// TIA Portal V17 export
// export: Created 2025-03-07T09:19:10.5525524Z, ExportSetting WithDefaults, DisplayName Totally Integrated Automation Portal, DisplayVersion V17 Update 8, DisplayName TIA Portal Openness, DisplayVersion V17 Update 8, DisplayName TIA Portal Version Control Interface, DisplayVersion V17, DisplayName SINAMICS Startdrive Advanced, DisplayVersion V17 SP2, DisplayName SINAMICS Startdrive G110M, G120, G120C, G120D, G120P, G115D, DisplayVersion V17 SP2, DisplayName SINAMICS Startdrive G130, G150, S120, S150, SINAMICS MV, S210, DisplayVersion V17 SP2, DisplayName STEP 7 Professional, DisplayVersion V17 Update 8, DisplayName SINUMERIK ONE STEP 7 Toolbox, DisplayVersion V17 Update 12, DisplayName SINUMERIK 840D sl STEP 7 Toolbox, DisplayVersion V17 Update 12, DisplayName STEP 7 Safety, DisplayVersion V17 Update 6, DisplayName WinCC Advanced, DisplayVersion V17 Update 8
FUNCTION "FC7201_HMI_DATA_FUNC" : Void   // FC7201, LAD
{ S7_Optimized_Access := 'FALSE' }
AUTHOR : ETXETAR
VERSION : 1.0
// stored: AutoNumber false, IsIECCheckEnabled false, SetENOAutomatically false, UDAEnableTagReadback false
   VAR_TEMP
      Sammel_1 : Bool;
      Sammel_2 : Bool;
      Sammel_3 : Bool;
      pin_main_table : Bool;
      main_table : Bool;
      Status1 : Int;
      Status2 : Int;
      sammel : Bool;
      aux1 : Bool;
      aux2 : Bool;
   END_VAR
   VAR_TEMP   // added for the SCL form of the ladder/FBD networks
      _w1 : Bool;
   END_VAR
BEGIN

REGION Network 1: AUTOMATIC
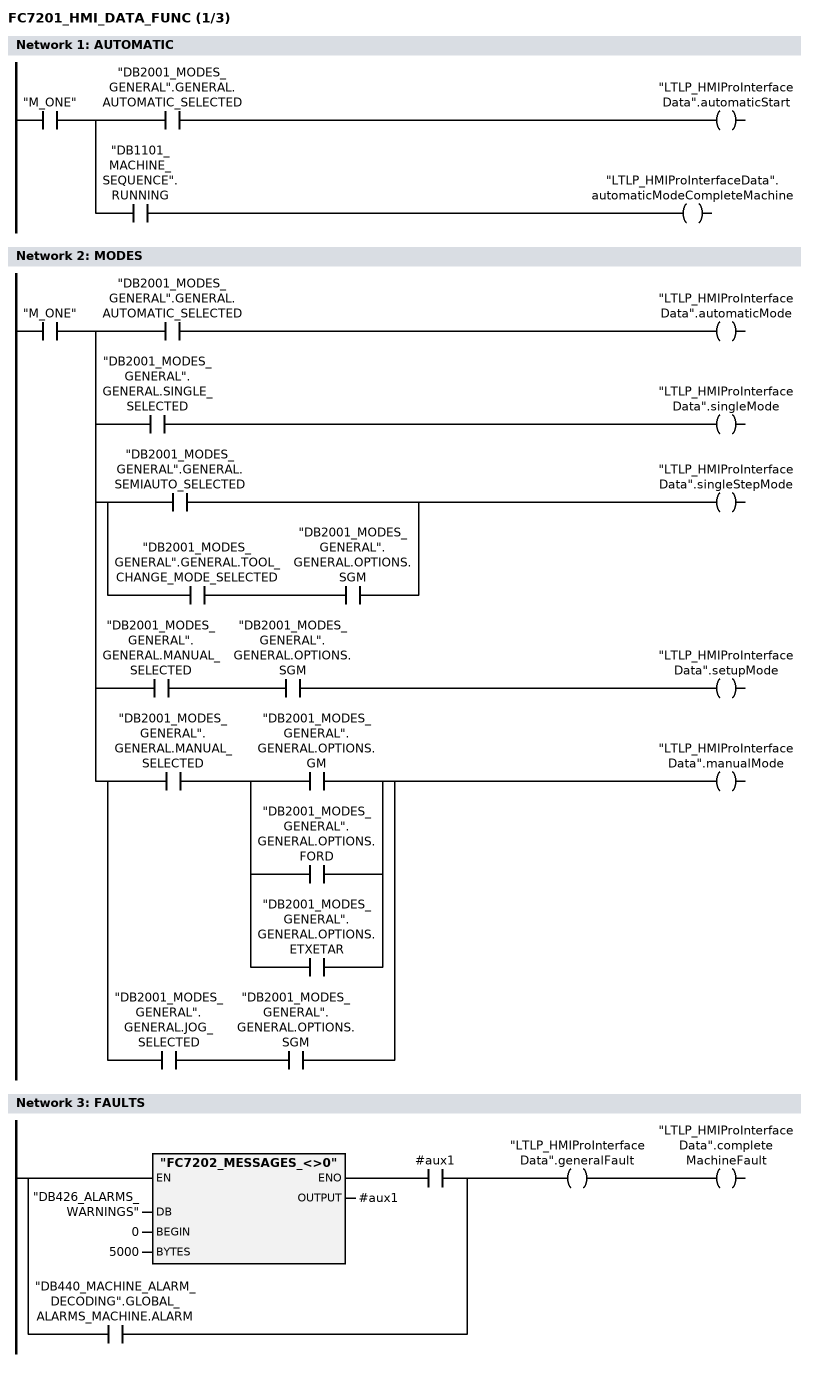
   RUNG wire#powerrail
      Contact( "M_ONE" )
      wire#w1
      Contact( "DB2001_MODES_GENERAL".GENERAL.AUTOMATIC_SELECTED )
      Coil( "LTLP_HMIProInterfaceData".automaticStart )
   END_RUNG
   RUNG wire#w1
      Contact( "DB1101_MACHINE_SEQUENCE".RUNNING )
      Coil( "LTLP_HMIProInterfaceData".automaticModeCompleteMachine )
   END_RUNG
   // the same network as SCL:
   "LTLP_HMIProInterfaceData".automaticStart := "M_ONE" AND "DB2001_MODES_GENERAL".GENERAL.AUTOMATIC_SELECTED;
   "LTLP_HMIProInterfaceData".automaticModeCompleteMachine := "M_ONE" AND "DB1101_MACHINE_SEQUENCE".RUNNING;
END_REGION

REGION Network 2: MODES
   RUNG wire#powerrail
      Contact( "M_ONE" )
      wire#w1
      Contact( "DB2001_MODES_GENERAL".GENERAL.AUTOMATIC_SELECTED )
      Coil( "LTLP_HMIProInterfaceData".automaticMode )
   END_RUNG
   RUNG wire#w1
      Contact( "DB2001_MODES_GENERAL".GENERAL.SINGLE_SELECTED )
      Coil( "LTLP_HMIProInterfaceData".singleMode )
   END_RUNG
   RUNG wire#w1
      Contact( "DB2001_MODES_GENERAL".GENERAL.SEMIAUTO_SELECTED )
      wire#w2
      Coil( "LTLP_HMIProInterfaceData".singleStepMode )
   END_RUNG
   RUNG wire#w1
      Contact( "DB2001_MODES_GENERAL".GENERAL.TOOL_CHANGE_MODE_SELECTED )
      Contact( "DB2001_MODES_GENERAL".GENERAL.OPTIONS.SGM )
   END_RUNG wire#w2
   RUNG wire#w1
      Contact( "DB2001_MODES_GENERAL".GENERAL.MANUAL_SELECTED )
      Contact( "DB2001_MODES_GENERAL".GENERAL.OPTIONS.SGM )
      Coil( "LTLP_HMIProInterfaceData".setupMode )
   END_RUNG
   RUNG wire#w1
      Contact( "DB2001_MODES_GENERAL".GENERAL.MANUAL_SELECTED )
      wire#w3
      Contact( "DB2001_MODES_GENERAL".GENERAL.OPTIONS.GM )
      wire#w4
      Coil( "LTLP_HMIProInterfaceData".manualMode )
   END_RUNG
   RUNG wire#w3
      Contact( "DB2001_MODES_GENERAL".GENERAL.OPTIONS.FORD )
   END_RUNG wire#w4
   RUNG wire#w3
      Contact( "DB2001_MODES_GENERAL".GENERAL.OPTIONS.ETXETAR )
   END_RUNG wire#w4
   RUNG wire#w1
      Contact( "DB2001_MODES_GENERAL".GENERAL.JOG_SELECTED )
      Contact( "DB2001_MODES_GENERAL".GENERAL.OPTIONS.SGM )
   END_RUNG wire#w4
   // the same network as SCL:
   "LTLP_HMIProInterfaceData".automaticMode := "M_ONE" AND "DB2001_MODES_GENERAL".GENERAL.AUTOMATIC_SELECTED;
   "LTLP_HMIProInterfaceData".singleMode := "M_ONE" AND "DB2001_MODES_GENERAL".GENERAL.SINGLE_SELECTED;
   "LTLP_HMIProInterfaceData".singleStepMode := "M_ONE" AND ("DB2001_MODES_GENERAL".GENERAL.SEMIAUTO_SELECTED OR ("DB2001_MODES_GENERAL".GENERAL.TOOL_CHANGE_MODE_SELECTED AND "DB2001_MODES_GENERAL".GENERAL.OPTIONS.SGM));
   "LTLP_HMIProInterfaceData".setupMode := "M_ONE" AND "DB2001_MODES_GENERAL".GENERAL.MANUAL_SELECTED AND "DB2001_MODES_GENERAL".GENERAL.OPTIONS.SGM;
   "LTLP_HMIProInterfaceData".manualMode := "M_ONE" AND (("DB2001_MODES_GENERAL".GENERAL.MANUAL_SELECTED AND ("DB2001_MODES_GENERAL".GENERAL.OPTIONS.GM OR "DB2001_MODES_GENERAL".GENERAL.OPTIONS.FORD OR "DB2001_MODES_GENERAL".GENERAL.OPTIONS.ETXETAR)) OR ("DB2001_MODES_GENERAL".GENERAL.JOG_SELECTED AND "DB2001_MODES_GENERAL".GENERAL.OPTIONS.SGM));
END_REGION

REGION Network 3: FAULTS
   RUNG wire#powerrail
      "FC7202_MESSAGES_<>0"(DB := "DB426_ALARMS_WARNINGS", "BEGIN" := 0, BYTES := 5000, OUTPUT => #aux1)
      Contact( #aux1 )
      wire#w1
      Coil( "LTLP_HMIProInterfaceData".generalFault )
      Coil( "LTLP_HMIProInterfaceData".completeMachineFault )
   END_RUNG
   RUNG wire#powerrail
      Contact( "DB440_MACHINE_ALARM_DECODING".GLOBAL_ALARMS_MACHINE.ALARM )
   END_RUNG wire#w1
   // the same network as SCL:
   "FC7202_MESSAGES_<>0"(DB := "DB426_ALARMS_WARNINGS",
                         "BEGIN" := 0,
                         BYTES := 5000,
                         OUTPUT => #aux1,
                         ENO => #_w1);
   "LTLP_HMIProInterfaceData".generalFault := (#_w1 AND #aux1) OR "DB440_MACHINE_ALARM_DECODING".GLOBAL_ALARMS_MACHINE.ALARM;
   "LTLP_HMIProInterfaceData".completeMachineFault := "LTLP_HMIProInterfaceData".generalFault;
END_REGION

REGION Network 4: WARNINGS
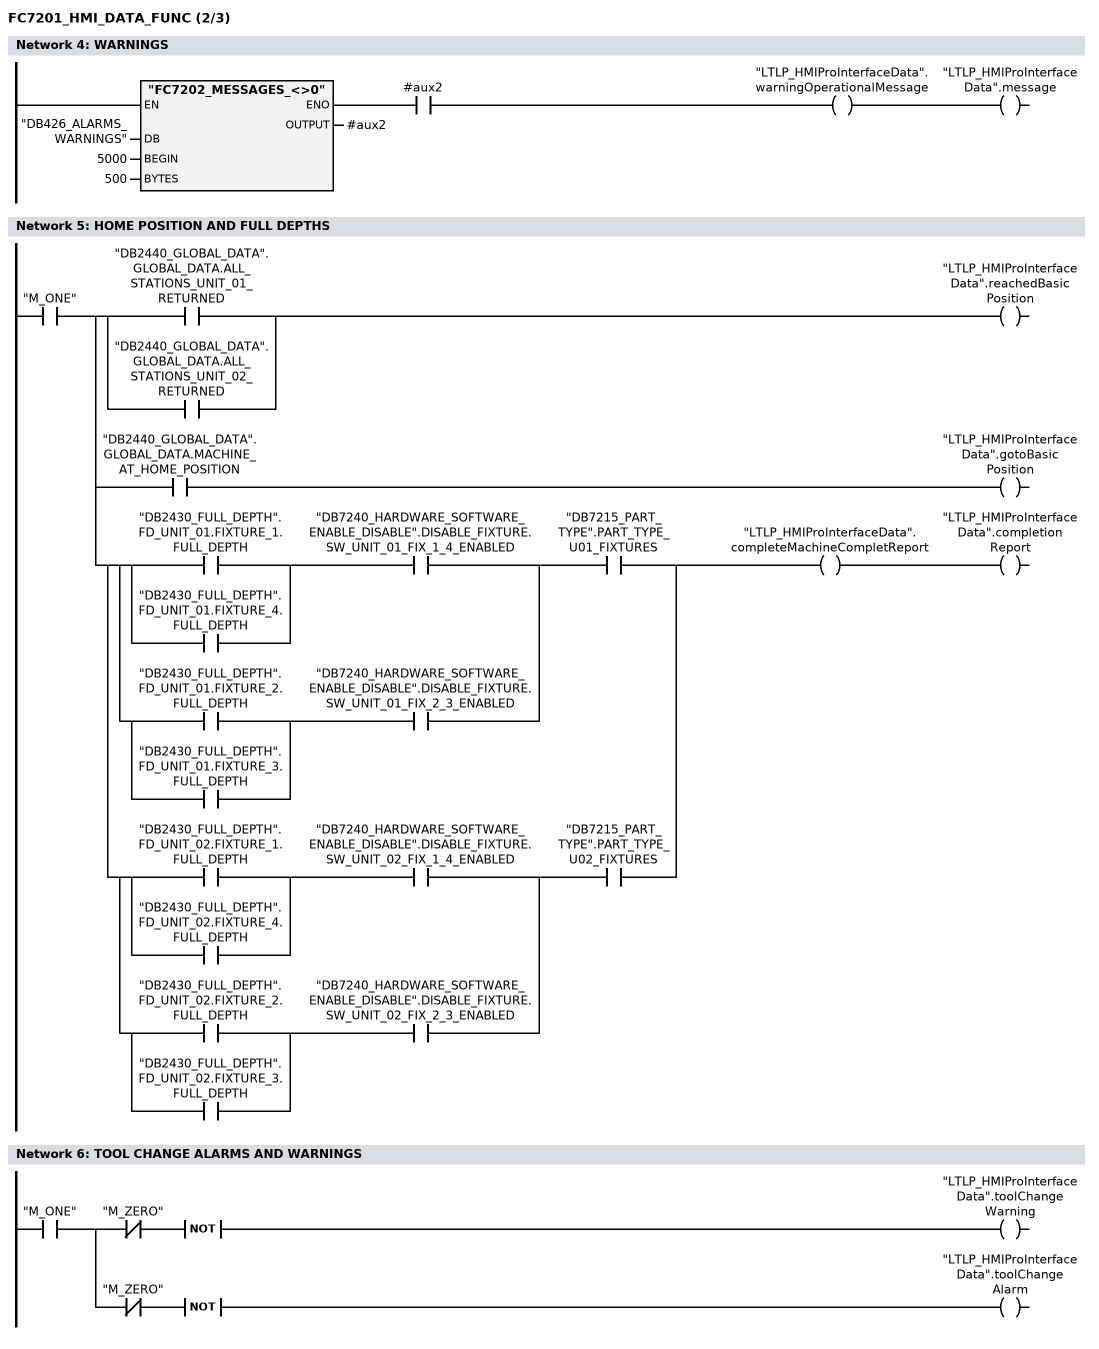
   RUNG wire#powerrail
      "FC7202_MESSAGES_<>0"(DB := "DB426_ALARMS_WARNINGS", "BEGIN" := 5000, BYTES := 500, OUTPUT => #aux2)
      Contact( #aux2 )
      Coil( "LTLP_HMIProInterfaceData".warningOperationalMessage )
      Coil( "LTLP_HMIProInterfaceData".message )
   END_RUNG
   // the same network as SCL:
   "FC7202_MESSAGES_<>0"(DB := "DB426_ALARMS_WARNINGS",
                         "BEGIN" := 5000,
                         BYTES := 500,
                         OUTPUT => #aux2,
                         ENO => #_w1);
   "LTLP_HMIProInterfaceData".warningOperationalMessage := #_w1 AND #aux2;
   "LTLP_HMIProInterfaceData".message := "LTLP_HMIProInterfaceData".warningOperationalMessage;
END_REGION

REGION Network 5: HOME POSITION AND FULL DEPTHS
   RUNG wire#powerrail
      Contact( "M_ONE" )
      wire#w1
      Contact( "DB2440_GLOBAL_DATA".GLOBAL_DATA.ALL_STATIONS_UNIT_01_RETURNED )
      wire#w2
      Coil( "LTLP_HMIProInterfaceData".reachedBasicPosition )
   END_RUNG
   RUNG wire#w1
      Contact( "DB2440_GLOBAL_DATA".GLOBAL_DATA.ALL_STATIONS_UNIT_02_RETURNED )
   END_RUNG wire#w2
   RUNG wire#w1
      Contact( "DB2440_GLOBAL_DATA".GLOBAL_DATA.MACHINE_AT_HOME_POSITION )
      Coil( "LTLP_HMIProInterfaceData".gotoBasicPosition )
   END_RUNG
   RUNG wire#w1
      Contact( "DB2430_FULL_DEPTH".FD_UNIT_01.FIXTURE_1.FULL_DEPTH )
      wire#w3
      Contact( "DB7240_HARDWARE_SOFTWARE_ENABLE_DISABLE".DISABLE_FIXTURE.SW_UNIT_01_FIX_1_4_ENABLED )
      wire#w4
      Contact( "DB7215_PART_TYPE".PART_TYPE_U01_FIXTURES )
      wire#w6
      Coil( "LTLP_HMIProInterfaceData".completeMachineCompletReport )
      Coil( "LTLP_HMIProInterfaceData".completionReport )
   END_RUNG
   RUNG wire#w1
      Contact( "DB2430_FULL_DEPTH".FD_UNIT_01.FIXTURE_4.FULL_DEPTH )
   END_RUNG wire#w3
   RUNG wire#w1
      Contact( "DB2430_FULL_DEPTH".FD_UNIT_01.FIXTURE_2.FULL_DEPTH )
      wire#w5
      Contact( "DB7240_HARDWARE_SOFTWARE_ENABLE_DISABLE".DISABLE_FIXTURE.SW_UNIT_01_FIX_2_3_ENABLED )
   END_RUNG wire#w4
   RUNG wire#w1
      Contact( "DB2430_FULL_DEPTH".FD_UNIT_01.FIXTURE_3.FULL_DEPTH )
   END_RUNG wire#w5
   RUNG wire#w1
      Contact( "DB2430_FULL_DEPTH".FD_UNIT_02.FIXTURE_1.FULL_DEPTH )
      wire#w7
      Contact( "DB7240_HARDWARE_SOFTWARE_ENABLE_DISABLE".DISABLE_FIXTURE.SW_UNIT_02_FIX_1_4_ENABLED )
      wire#w8
      Contact( "DB7215_PART_TYPE".PART_TYPE_U02_FIXTURES )
   END_RUNG wire#w6
   RUNG wire#w1
      Contact( "DB2430_FULL_DEPTH".FD_UNIT_02.FIXTURE_4.FULL_DEPTH )
   END_RUNG wire#w7
   RUNG wire#w1
      Contact( "DB2430_FULL_DEPTH".FD_UNIT_02.FIXTURE_2.FULL_DEPTH )
      wire#w9
      Contact( "DB7240_HARDWARE_SOFTWARE_ENABLE_DISABLE".DISABLE_FIXTURE.SW_UNIT_02_FIX_2_3_ENABLED )
   END_RUNG wire#w8
   RUNG wire#w1
      Contact( "DB2430_FULL_DEPTH".FD_UNIT_02.FIXTURE_3.FULL_DEPTH )
   END_RUNG wire#w9
   // the same network as SCL:
   "LTLP_HMIProInterfaceData".reachedBasicPosition := "M_ONE" AND ("DB2440_GLOBAL_DATA".GLOBAL_DATA.ALL_STATIONS_UNIT_01_RETURNED OR "DB2440_GLOBAL_DATA".GLOBAL_DATA.ALL_STATIONS_UNIT_02_RETURNED);
   "LTLP_HMIProInterfaceData".gotoBasicPosition := "M_ONE" AND "DB2440_GLOBAL_DATA".GLOBAL_DATA.MACHINE_AT_HOME_POSITION;
   "LTLP_HMIProInterfaceData".completeMachineCompletReport := "M_ONE" AND ((((("DB2430_FULL_DEPTH".FD_UNIT_01.FIXTURE_1.FULL_DEPTH OR "DB2430_FULL_DEPTH".FD_UNIT_01.FIXTURE_4.FULL_DEPTH) AND "DB7240_HARDWARE_SOFTWARE_ENABLE_DISABLE".DISABLE_FIXTURE.SW_UNIT_01_FIX_1_4_ENABLED) OR (("DB2430_FULL_DEPTH".FD_UNIT_01.FIXTURE_2.FULL_DEPTH OR "DB2430_FULL_DEPTH".FD_UNIT_01.FIXTURE_3.FULL_DEPTH) AND "DB7240_HARDWARE_SOFTWARE_ENABLE_DISABLE".DISABLE_FIXTURE.SW_UNIT_01_FIX_2_3_ENABLED)) AND "DB7215_PART_TYPE".PART_TYPE_U01_FIXTURES) OR (((("DB2430_FULL_DEPTH".FD_UNIT_02.FIXTURE_1.FULL_DEPTH OR "DB2430_FULL_DEPTH".FD_UNIT_02.FIXTURE_4.FULL_DEPTH) AND "DB7240_HARDWARE_SOFTWARE_ENABLE_DISABLE".DISABLE_FIXTURE.SW_UNIT_02_FIX_1_4_ENABLED) OR (("DB2430_FULL_DEPTH".FD_UNIT_02.FIXTURE_2.FULL_DEPTH OR "DB2430_FULL_DEPTH".FD_UNIT_02.FIXTURE_3.FULL_DEPTH) AND "DB7240_HARDWARE_SOFTWARE_ENABLE_DISABLE".DISABLE_FIXTURE.SW_UNIT_02_FIX_2_3_ENABLED)) AND "DB7215_PART_TYPE".PART_TYPE_U02_FIXTURES));
   "LTLP_HMIProInterfaceData".completionReport := "LTLP_HMIProInterfaceData".completeMachineCompletReport;
END_REGION

REGION Network 6: TOOL CHANGE ALARMS AND WARNINGS
   RUNG wire#powerrail
      Contact( "M_ONE" )
      wire#w1
      I_Contact( "M_ZERO" )
      Not()
      Coil( "LTLP_HMIProInterfaceData".toolChangeWarning )
   END_RUNG
   RUNG wire#w1
      I_Contact( "M_ZERO" )
      Not()
      Coil( "LTLP_HMIProInterfaceData".toolChangeAlarm )
   END_RUNG
   // the same network as SCL:
   "LTLP_HMIProInterfaceData".toolChangeWarning := NOT ("M_ONE" AND NOT "M_ZERO");
   "LTLP_HMIProInterfaceData".toolChangeAlarm := NOT ("M_ONE" AND NOT "M_ZERO");
END_REGION

REGION Network 7: HMI HEADER
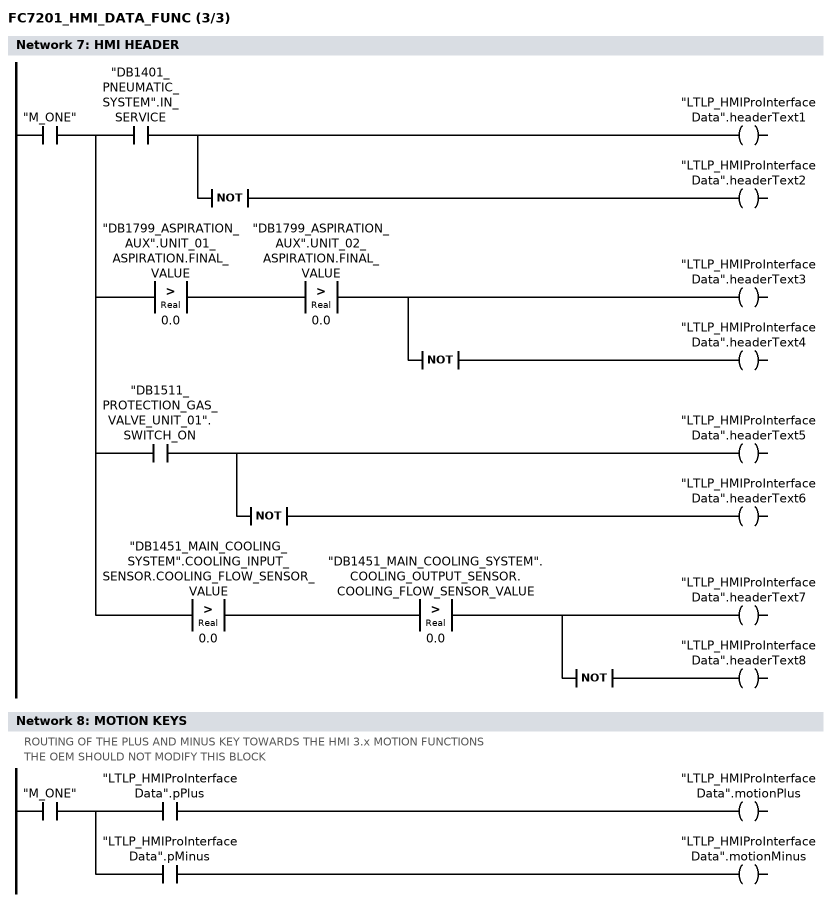
   RUNG wire#powerrail
      Contact( "M_ONE" )
      wire#w1
      Contact( "DB1401_PNEUMATIC_SYSTEM".IN_SERVICE )
      wire#w2
      Coil( "LTLP_HMIProInterfaceData".headerText1 )
   END_RUNG
   RUNG wire#w2
      Not()
      Coil( "LTLP_HMIProInterfaceData".headerText2 )
   END_RUNG
   RUNG wire#w1
      { S7_Templates := "SrcType := Real" } GT_Contact(in1 := "DB1799_ASPIRATION_AUX".UNIT_01_ASPIRATION.FINAL_VALUE, in2 := 0.0)
      { S7_Templates := "SrcType := Real" } GT_Contact(in1 := "DB1799_ASPIRATION_AUX".UNIT_02_ASPIRATION.FINAL_VALUE, in2 := 0.0)
      wire#w3
      Coil( "LTLP_HMIProInterfaceData".headerText3 )
   END_RUNG
   RUNG wire#w3
      Not()
      Coil( "LTLP_HMIProInterfaceData".headerText4 )
   END_RUNG
   RUNG wire#w1
      Contact( "DB1511_PROTECTION_GAS_VALVE_UNIT_01".SWITCH_ON )
      wire#w4
      Coil( "LTLP_HMIProInterfaceData".headerText5 )
   END_RUNG
   RUNG wire#w4
      Not()
      Coil( "LTLP_HMIProInterfaceData".headerText6 )
   END_RUNG
   RUNG wire#w1
      { S7_Templates := "SrcType := Real" } GT_Contact(in1 := "DB1451_MAIN_COOLING_SYSTEM".COOLING_INPUT_SENSOR.COOLING_FLOW_SENSOR_VALUE, in2 := 0.0)
      { S7_Templates := "SrcType := Real" } GT_Contact(in1 := "DB1451_MAIN_COOLING_SYSTEM".COOLING_OUTPUT_SENSOR.COOLING_FLOW_SENSOR_VALUE, in2 := 0.0)
      wire#w5
      Coil( "LTLP_HMIProInterfaceData".headerText7 )
   END_RUNG
   RUNG wire#w5
      Not()
      Coil( "LTLP_HMIProInterfaceData".headerText8 )
   END_RUNG
   // the same network as SCL:
   "LTLP_HMIProInterfaceData".headerText1 := "M_ONE" AND "DB1401_PNEUMATIC_SYSTEM".IN_SERVICE;
   "LTLP_HMIProInterfaceData".headerText2 := NOT "LTLP_HMIProInterfaceData".headerText1;
   "LTLP_HMIProInterfaceData".headerText3 := "M_ONE" AND ("DB1799_ASPIRATION_AUX".UNIT_01_ASPIRATION.FINAL_VALUE > 0.0) AND ("DB1799_ASPIRATION_AUX".UNIT_02_ASPIRATION.FINAL_VALUE > 0.0);
   "LTLP_HMIProInterfaceData".headerText4 := NOT "LTLP_HMIProInterfaceData".headerText3;
   "LTLP_HMIProInterfaceData".headerText5 := "M_ONE" AND "DB1511_PROTECTION_GAS_VALVE_UNIT_01".SWITCH_ON;
   "LTLP_HMIProInterfaceData".headerText6 := NOT "LTLP_HMIProInterfaceData".headerText5;
   "LTLP_HMIProInterfaceData".headerText7 := "M_ONE" AND ("DB1451_MAIN_COOLING_SYSTEM".COOLING_INPUT_SENSOR.COOLING_FLOW_SENSOR_VALUE > 0.0) AND ("DB1451_MAIN_COOLING_SYSTEM".COOLING_OUTPUT_SENSOR.COOLING_FLOW_SENSOR_VALUE > 0.0);
   "LTLP_HMIProInterfaceData".headerText8 := NOT "LTLP_HMIProInterfaceData".headerText7;
END_REGION

REGION Network 8: MOTION KEYS
   // ROUTING OF THE PLUS AND MINUS KEY TOWARDS THE HMI 3.x MOTION FUNCTIONS
   // THE OEM SHOULD NOT MODIFY THIS BLOCK
   RUNG wire#powerrail
      Contact( "M_ONE" )
      wire#w1
      Contact( "LTLP_HMIProInterfaceData".pPlus )
      Coil( "LTLP_HMIProInterfaceData".motionPlus )
   END_RUNG
   RUNG wire#w1
      Contact( "LTLP_HMIProInterfaceData".pMinus )
      Coil( "LTLP_HMIProInterfaceData".motionMinus )
   END_RUNG
   // the same network as SCL:
   "LTLP_HMIProInterfaceData".motionPlus := "M_ONE" AND "LTLP_HMIProInterfaceData".pPlus;
   "LTLP_HMIProInterfaceData".motionMinus := "M_ONE" AND "LTLP_HMIProInterfaceData".pMinus;
END_REGION
END_FUNCTION
